FUNCTION_BLOCK FB_Cylinder_ExtendedSensor EXTENDS FB_CylinderBase
VAR_INPUT
END_VAR
VAR_OUTPUT
END_VAR
VAR
	fbExtendedSensor			: FB_Sensor;
END_VAR

METHOD HardwareUpdate : BOOL
VAR_INPUT
END_VAR
fbSimExtend_TON();		//Call timer FB
fbSimRetract_TON();		//Call timer FB

GenerateFeedback(bExtend := bExtendCommand,
				 bRetract := bRetractCommand,
				 bExtended_Generated => ,
				 bRetracted_Generated => bRetractedFeedback);
bExtendedFeedback := fbExtendedSensor.Active;
END_METHOD

END_FUNCTION_BLOCK

(* stored: Version 1.1.0.1, ProductVersion 3.1.4024.9
   POU FB_Cylinder_ExtendedSensor: Id {e2d251e8-bd09-49e4-9ebd-44d33b58dd3d}, SpecialFunc None
   Folder 01_SUPER_Overrides: Id {cff9f11a-9033-4a5f-a661-5bb32e064a1f}
   Method HardwareUpdate: Id {e1108088-0470-4f28-a4d4-fdb757cbab79} *)
